(*			
	RAFALOS
	Rafał Osajda		19.09.2025		TC 4024.66
	Rodzic dla wszystkich podzespołów głównych w maszynie 
*)
FUNCTION_BLOCK FB_BaseMainComponent EXTENDS FB_BaseComplexElement IMPLEMENTS ITF_BaseMainComponent, ITF_BaseMainComponent_HMI_Connector
VAR
END_VAR

END_FUNCTION_BLOCK

(* stored: Version 1.1.0.1
   POU FB_BaseMainComponent: Id {b23ea2e3-7979-0bc9-362e-7cf0941731d6}, SpecialFunc None *)
